INTERFACE I_HostInputPorts EXTENDS __SYSTEM.IQueryInterface

PROPERTY InputPorts : I_InputPorts
GET
END_GET
END_PROPERTY

END_INTERFACE

(* stored: Version 1.1.0.1, ProductVersion 3.1.4024.12
   Itf I_HostInputPorts: Id {83257efe-17cc-4986-a355-19d5cde0900d}
   Property InputPorts: Id {3145f9b9-d962-446c-83c0-6a1f53f8850c}
   Get Get: Id {79cbc02b-3dc0-4d10-b1b3-2dab536a3d36} *)
